Fanuc TP program (LS listing): HOME_SAFE.ls

/PROG HOME_SAFE
/ATTR
OWNER		= MNEDITOR;
COMMENT		= "Study drill. FANUC rights. Educational; own risk.";
PROG_SIZE	= 0;
CREATE		= DATE 26-08-20  TIME 20:00:00;
MODIFIED	= DATE 26-08-20  TIME 20:00:00;
FILE_NAME	= ;
VERSION		= 0;
LINE_COUNT	= 12;
MEMORY_SIZE	= 0;
PROTECT		= READ_WRITE;
TCD:  STACK_SIZE	= 0,
      TASK_PRIORITY	= 50,
      TIME_SLICE	= 0,
      BUSY_LAMP_OFF	= 0,
      ABORT_REQUEST	= 0,
      PAUSE_REQUEST	= 0;
DEFAULT_GROUP	= 1,*,*,*,*;
CONTROL_CODE	= 00000000 00000000;
/APPL
/MN
   0:  ! FANUC retains all rights in its marks/software/manuals. Educational only. Use at your own consent and risk. See LEGAL.md ;
   1:  ! SAMPLE ONLY - replace frames I/O home with cell data ;
   2:  ! Ask: model controller pendant EOAT UTOOL UFRAME home ;
   3:  UFRAME_NUM=1 ;
   4:  UTOOL_NUM=1 ;
   5:  ! PR[1:Home] must be taught on the real robot ;
   6:  J PR[1:Home] 20% FINE    ;
   7:  ! Optional DO handshake - numbers are PLACEHOLDERS ;
   8:  ! DO[101:AtHome]=ON ;
   9:  END ;
/POS
/END
